(* IEC 61131-3 sources: volt/packages/volt-lsp-iec/test-corpus/bakon-nano/Device/Plc Logic/Application/POUs/RecipeManagement, 4 files *)

(* ---- L_RecipeManager.pou ---- *)
FUNCTION_BLOCK L_RecipeManager
VAR_INPUT
	xEnable					: BOOL;				//Enable functions
	sDatabaseName			: STRING;			//Database of recipe manager (name)
	sRecipeName				: STRING;			//Selected recipe (name)
END_VAR
VAR_IN_OUT
	xRecipe_Delete			: BOOL;				//Delete definition (DeleteRecipeFile)
	xRecipe_Load			: BOOL;				//Load recipe (LoadAndWriteRecipe)
	xRecipe_Save			: BOOL;				//Save recipe (ReadAndSaveRecipe)
	xRecipe_SaveAs			: BOOL;				//Save recipe (ReadAndSaveRecipe)
	sActiveRecipe			: STRING;			//Active machine recipe
END_VAR
VAR_OUTPUT
	xEnabled				: BOOL;				//Function enabled
	iNumberOfRecipes		: INT;				//Counted recipes in database
	sRecipeNames			: STRING(gc_iSizeRecipesNames);	//Combined recipe names
	dwReturnValue			: DWORD;			//Return value of recipe manager
END_VAR

VAR
	RecipeHandler			: RecipeManCommands;//Function to access PLC recipes
	sRecipeLocal			: STRING;			//Used to concat
	psNames					: POINTER TO STRING(gc_iSizeRecipesNames);
	psLocal					: POINTER TO STRING;
	iLoopNames				: INT;				//Loop recipe names
	strSearchChar			: STRING;
	iResult					: INT;
END_VAR
VAR CONSTANT
	gc_iSizeRecipesNames 	: INT := 5000;
	//gc_iMaxResultsFinder	: INT := 10;
END_VAR
%LANGUAGE ST
IF xEnable THEN
	xEnabled := xEnable;
	//************************************************************************Refresh data
	//Get data addresses
	psNames := ADR(sRecipeNames);
	psLocal := ADR(sRecipeLocal);
	//Refresh file buffer
	RecipeHandler.ReloadRecipes(sDatabaseName);
	//Get recipe count
	iNumberOfRecipes := RecipeHandler.GetRecipeCount(sDatabaseName);
	//Get saved recipe informations
	sRecipeNames:='';
	FOR iLoopNames:=0 TO iNumberOfRecipes-1 BY 1 DO
		//Get recipe name
		sRecipeLocal := '';
		RecipeHandler.GetRecipeNames(sDatabaseName, ADR(sRecipeLocal) , 1, iLoopNames);

		//Add recipe name to end of string
		StrConcatA(pstFrom:= psLocal, pstTo:= psNames, iBufferSize:= gc_iSizeRecipesNames);

		//Add seperator to end
		sRecipeLocal := ';';
		StrConcatA(pstFrom:= psLocal, pstTo:= psNames, iBufferSize:= gc_iSizeRecipesNames);
	END_FOR

	//************************************************************************Load recipe to HMI
	IF xRecipe_Load THEN
		dwReturnValue:=RecipeHandler.LoadAndWriteRecipe(sDatabaseName, sRecipeName);//Load to handler recipe
		IF dwReturnValue = 0 THEN
			sActiveRecipe := sRecipeName;
		END_IF
		xRecipe_Load:=FALSE;
	END_IF
	//************************************************************************Save recipe to database
	IF xRecipe_Save THEN
		dwReturnValue:=RecipeHandler.ReadAndSaveRecipe(sDatabaseName, sActiveRecipe);		//Save to file
		xRecipe_Save := FALSE;
	END_IF
	//************************************************************************Delete recipe
	//More than 0 recipes left
	IF xRecipe_Delete THEN
		dwReturnValue:=RecipeHandler.DeleteRecipe(sDatabaseName, sRecipeName);	//Remove database link
		IF sActiveRecipe = sRecipeName THEN
			sActiveRecipe:='';
		END_IF
		xRecipe_Delete := FALSE;
	END_IF
	//************************************************************************Save recipe as
	IF xRecipe_SaveAs THEN
		strSearchChar:='.';
		iResult:=StrFindA(pst1:=ADR(sRecipeName) , pst2:= ADR(strSearchChar), uiSearchStart:= 0);
		IF iResult <> 0 THEN
			dwReturnValue:=16#7000;
			RETURN;
		END_IF

		dwReturnValue:=RecipeHandler.CreateRecipe(sDatabaseName, sRecipeName);		//Create new file and save

		//New recipe OR when recipe already existed
		IF dwReturnValue = 16#4005 OR dwReturnValue = 0 THEN
			dwReturnValue:=RecipeHandler.ReadAndSaveRecipe(sDatabaseName, sRecipeName);	//Create new file and save
		END_IF
		IF dwReturnValue = 0 THEN
			dwReturnValue:=RecipeHandler.LoadAndWriteRecipe(sDatabaseName, sRecipeName);//Load to handler recipe
			dwReturnValue:=SEL(dwReturnValue <> 0, 0, 16#7001);
		END_IF
		IF dwReturnValue = 0 THEN
			sActiveRecipe := sRecipeName;
		END_IF
		xRecipe_SaveAs := FALSE;
	END_IF

ELSE
	sActiveRecipe := '';
	dwReturnValue:=0;
END_IF

END_FUNCTION_BLOCK

(* ---- L_RecipeManager_Rcp.pou ---- *)
FUNCTION_BLOCK L_RecipeManager_Rcp
VAR_INPUT
	xEnable						: BOOL;				//Enable functions
	sDatabaseName				: STRING;			//Database of recipe manager (name)
END_VAR
VAR_IN_OUT
	sSelectedRecipeName			: STRING;
	xRecipe_Load				: BOOL;
	xRecipe_New					: BOOL;
	xRecipe_Edit				: BOOL;
	xRecipe_Save				: BOOL;
	xRecipe_Copy				: BOOL;
	xRecipe_Delete				: BOOL;
	xRecipe_Update				: BOOL;
	scRecipeVisu				: sMACH_RCP_Parameters;
	scRecipePLC					: sMACH_RCP_Parameters;
END_VAR
VAR_OUTPUT
	xEnabled					: BOOL;				//Function enabled
	iNumberOfRecipes			: INT;				//Counted recipes in database
	sRecipeNames				: STRING(gc_iSizeRecipesNames);	//Combined recipe names
	dwReturnValue				: DWORD;			//Return value of recipe manager
END_VAR
VAR
	RecipeHandler				: RecipeManCommands;//Function to access PLC recipes
	sRecipeLocal				: STRING;			//Used to concat
	psNames						: POINTER TO STRING(gc_iSizeRecipesNames);
	psLocal						: POINTER TO STRING;
	iLoopNames					: INT;				//Loop recipe names
	strSearchChar				: STRING;
	iResult						: INT;
	sRecipNameTemp: STRING;
END_VAR
VAR CONSTANT
	gc_iSizeRecipesNames 		: INT := 16384;
END_VAR
%LANGUAGE ST
IF xEnable THEN
	xEnabled := xEnable;
	//************************************************************************Refresh data
	//Get data addresses
	psNames := ADR(sRecipeNames);
	psLocal := ADR(sRecipeLocal);
	//Refresh file buffer
	RecipeHandler.ReloadRecipes(sDatabaseName);
	//Get recipe count
	iNumberOfRecipes := RecipeHandler.GetRecipeCount(sDatabaseName);
	//Get saved recipe informations
	sRecipeNames:='';
	FOR iLoopNames:=0 TO iNumberOfRecipes-1 BY 1 DO
		//Get recipe name
		sRecipeLocal := '';
		RecipeHandler.GetRecipeNames(sDatabaseName, ADR(sRecipeLocal) , 1, iLoopNames);

		//Add recipe name to end of string
		StrConcatA(pstFrom:= psLocal, pstTo:= psNames, iBufferSize:= gc_iSizeRecipesNames);

		//Add seperator to end
		sRecipeLocal := ';';
		StrConcatA(pstFrom:= psLocal, pstTo:= psNames, iBufferSize:= gc_iSizeRecipesNames);
	END_FOR
	IF xRecipe_Load THEN
		dwReturnValue:=RecipeHandler.LoadAndWriteRecipe(sDatabaseName, sSelectedRecipeName);//Load to handler recipe
		IF dwReturnValue = 0 THEN
			scRecipePLC:=scRecipeVisu;
		END_IF
		xRecipe_Load:=FALSE;
	END_IF
	IF xRecipe_New THEN
		strSearchChar:='.';
		dwReturnValue:=INT_TO_DWORD(StrFindA(pst1:=ADR(scRecipeVisu.sRecipeName) , pst2:= ADR(strSearchChar), uiSearchStart:= 0));
		IF dwReturnValue = 0 THEN
			dwReturnValue:=RecipeHandler.CreateRecipe(sDatabaseName, scRecipeVisu.sRecipeName);
		ELSE
			dwReturnValue:=16#7000;
		END_IF
		xRecipe_New := FALSE;
	END_IF
	IF xRecipe_Edit THEN
		dwReturnValue:=RecipeHandler.LoadAndWriteRecipe(sDatabaseName, sSelectedRecipeName);//Load to handler recipe
		xRecipe_Edit:=FALSE;
	END_IF
	IF xRecipe_Save THEN
		dwReturnValue:=RecipeHandler.ReadAndSaveRecipe(sDatabaseName, scRecipeVisu.sRecipeName);	//Create new file and save
		xRecipe_Save := FALSE;
	END_IF
	IF xRecipe_Copy THEN
		sRecipNameTemp:=scRecipeVisu.sRecipeName;
		dwReturnValue:=RecipeHandler.LoadAndWriteRecipe(sDatabaseName, sSelectedRecipeName);
		scRecipeVisu.sRecipeName:=sRecipNameTemp;
		strSearchChar:='.';
		dwReturnValue:=INT_TO_DWORD(StrFindA(pst1:=ADR(scRecipeVisu.sRecipeName) , pst2:= ADR(strSearchChar), uiSearchStart:= 0));
		IF dwReturnValue = 0 THEN
			dwReturnValue:=RecipeHandler.CreateRecipe(sDatabaseName, scRecipeVisu.sRecipeName);
		ELSE
			dwReturnValue:=16#7000;
		END_IF
		xRecipe_Copy := FALSE;
	END_IF
	IF xRecipe_Delete THEN
		dwReturnValue:=RecipeHandler.DeleteRecipe(sDatabaseName, sSelectedRecipeName);	//Remove database link
		xRecipe_Delete := FALSE;
	END_IF
	IF xRecipe_Update THEN
		scRecipeVisu:=scRecipePLC;
		dwReturnValue:=RecipeHandler.ReadAndSaveRecipe(sDatabaseName, scRecipeVisu.sRecipeName);	//Create new file and save
		xRecipe_Update := FALSE;
	END_IF
ELSE
	dwReturnValue:=0;
END_IF

END_FUNCTION_BLOCK

(* ---- RCP_RecipeHandler.pou ---- *)
PROGRAM RCP_RecipeHandler
VAR
	{warning 'Disabled for compatibility SVE'}
	//DiffLogger								: DifferenceLogger;
	bOldRect : BOOL;
	bOldEight : BOOL;
END_VAR
%LANGUAGE ST
(*Reset recipe*)
IF		g_HMI_MachCommand.CMD.bResetRecipe
THEN

		g_HMI_RCP_Parameters.nProductType				:= Prod_Tray_Rectangle_1x1;
		g_HMI_RCP_Parameters.rStartHeightKnife			:= 60;		(* Starthoogte, gemeten vanaf onderzijde mes tot aan de tafel *)
		g_HMI_RCP_Parameters.rStopHeightKnife			:= 0;		(* Stophoogte, gemeten vanaf onderzijde mes tot aan de tafel *)
		g_HMI_RCP_Parameters.nPartsRound				:= 12;			(*aantal stukken ronde taart *)
		g_HMI_RCP_Parameters.nPartsX					:= 5;			(*aantal stukken in X richting*)
		g_HMI_RCP_Parameters.nPartsY					:= 5;			(*aantal stukken in Y richting*)
		g_HMI_RCP_Parameters.rAngleInDegrees			:= 55;		(* Angle in degrees when producttype is diagonal *)
		g_HMI_RCP_Parameters.rProdLength_InX			:= 500;		(* Size of slab in line with the belt*)
		g_HMI_RCP_Parameters.rProdLength_InY			:= 300;		(* Size of slab perpendicular to the belt*)
		g_HMI_RCP_Parameters.rUSHeightStart			:= 60;		(* Start height ultrasonic generator (position Z-axis) *)
		g_HMI_RCP_Parameters.rUSHeightStop			:= 60;		(* Stop height ultrasonic generator (position Z-axis) *)
		g_HMI_RCP_Parameters.dwUltrasonicPower1		:= 50;
		g_HMI_RCP_Parameters.rCutSpeedZ_Down1		:= 50;			(* neergaande snelheid boven product in %*)
		g_HMI_RCP_Parameters.rCutSpeedZ_Down2		:= 50;			(* neergaande snelheid in het product in %*)
		g_HMI_RCP_Parameters.rCutSpeedZ_Up1			:= 50;			(* opgaande snelheid in het product in %*)
		g_HMI_RCP_Parameters.rSizeTrimRight			:= 8;		(*grootte van de afvalrand in de X richting aan de rechterzijde*)
		g_HMI_RCP_Parameters.rSizeTrimLeft			:= 8;		(*grootte van de afvalrand in de X richting aan de linkerzijde*)
		g_HMI_RCP_Parameters.rSizeTrimRear				:= 8;		(*grootte van de afvalrand in de Y richting aan de achterzijde*)
		g_HMI_RCP_Parameters.rSizeTrimFront			:= 8;		(*grootte van de afvalrand in de Y richting aan de voorzijde*)
		g_HMI_RCP_Parameters.rMidPosOffsetRound1X	:= 0;		(* For round products *)
		g_HMI_RCP_Parameters.rMidPosOffsetRound1Y	:= 0;		(* For round products *)
		g_HMI_RCP_Parameters.rMidPosOffsetRound2X	:= 0;		(* For round products *)
		g_HMI_RCP_Parameters.rMidPosOffsetRound2Y	:= 0;		(* For round products *)
		g_HMI_RCP_Parameters.bUseRectanglesForTriangles	:= FALSE;	(* For triangles only *)
		g_HMI_RCP_Parameters.rPartSizeX					:= 50;		(* For triangles only *)
		g_HMI_RCP_Parameters.rPartSizeY					:= 50;		(* For triangles only *)
		g_HMI_RCP_Parameters.rShiftCompensation		:= 0;

		g_HMI_MachCommand.CMD.bResetRecipe		:= FALSE;
		g_HMI_bRecipeIsReset								:= TRUE;

END_IF

(* Recept variabele driehoek in tray resetten indien deze keuze niet gemaakt is in de product optie pagina *)
IF NOT g_HMI_dwProductOptions.15 THEN
	g_HMI_RCP_Parameters.bTrianglesInTray := FALSE;
END_IF

(*Afvalrand limieten bepalen*) (*Minimaal een stuk van 10mm overhouden, maximale afvalrand van 500*)
CASE G_HMI_RCP_Parameters.nProductType OF
	Prod_Slab_Rectangle_1x1, Prod_Slab_Triangle_1x1, Prod_Slab_Diagonal_1x1, Prod_Slab_Rectangle_1x1_Clamp:	(*Slab products*)
	g_sHMI_Mach_UnitStatus.rWasteFrontMax 	:= MIN(500,(g_HMI_RCP_Parameters.rProdLength_InY - 10 - g_HMI_RCP_Parameters.rSizeTrimRear));
	g_sHMI_Mach_UnitStatus.rWasteRearMax 	:= MIN(500,(g_HMI_RCP_Parameters.rProdLength_InY - 10 - g_HMI_RCP_Parameters.rSizeTrimFront));
	g_sHMI_Mach_UnitStatus.rWasteRightMax 	:= MIN(500,(g_HMI_RCP_Parameters.rProdLength_InX - 10 - g_HMI_RCP_Parameters.rSizeTrimLeft));
	g_sHMI_Mach_UnitStatus.rWasteLeftMax 	:= MIN(500,(g_HMI_RCP_Parameters.rProdLength_InX - 10 - g_HMI_RCP_Parameters.rSizeTrimRight));

	Prod_Tray_Rectangle_1x2		:		(* ProductType = 4 = Tray Square Small *)
	g_sHMI_Mach_UnitStatus.rWasteFrontMax 	:= MIN(500,(g_HMI_MCH_Parameters.rProdLengthTraySmall_InY - 10 - g_HMI_RCP_Parameters.rSizeTrimRear));
	g_sHMI_Mach_UnitStatus.rWasteRearMax 	:= MIN(500,(g_HMI_MCH_Parameters.rProdLengthTraySmall_InY - 10 - g_HMI_RCP_Parameters.rSizeTrimFront));
	g_sHMI_Mach_UnitStatus.rWasteRightMax 	:= MIN(500,(g_HMI_MCH_Parameters.rProdLengthTraySmall_InX - 10 - g_HMI_RCP_Parameters.rSizeTrimLeft));
	g_sHMI_Mach_UnitStatus.rWasteLeftMax 	:= MIN(500,(g_HMI_MCH_Parameters.rProdLengthTraySmall_InX - 10 - g_HMI_RCP_Parameters.rSizeTrimRight));

	Prod_Tray_Rectangle_1x1		:		(* ProductType = 5 = Tray Square Large *)
	g_sHMI_Mach_UnitStatus.rWasteFrontMax 	:= MIN(500,(g_HMI_MCH_Parameters.rProdLengthTrayLarge_InY - 10 - g_HMI_RCP_Parameters.rSizeTrimRear));
	g_sHMI_Mach_UnitStatus.rWasteRearMax 	:= MIN(500,(g_HMI_MCH_Parameters.rProdLengthTrayLarge_InY - 10 - g_HMI_RCP_Parameters.rSizeTrimFront));
	g_sHMI_Mach_UnitStatus.rWasteRightMax 	:= MIN(500,(g_HMI_MCH_Parameters.rProdLengthTrayLarge_InX - 10 - g_HMI_RCP_Parameters.rSizeTrimLeft));
	g_sHMI_Mach_UnitStatus.rWasteLeftMax 	:= MIN(500,(g_HMI_MCH_Parameters.rProdLengthTrayLarge_InX - 10 - g_HMI_RCP_Parameters.rSizeTrimRight));

	Prod_Tray_Rectangle_1x4		:		(* ProductType = 6 = Tray Square 4 on a table *)
	g_sHMI_Mach_UnitStatus.rWasteFrontMax 	:= MIN(500,(g_HMI_MCH_Parameters.rProdLengthTrayTriple_InY - 10 - g_HMI_RCP_Parameters.rSizeTrimRear));
	g_sHMI_Mach_UnitStatus.rWasteRearMax 	:= MIN(500,(g_HMI_MCH_Parameters.rProdLengthTrayTriple_InY - 10 - g_HMI_RCP_Parameters.rSizeTrimFront));
	g_sHMI_Mach_UnitStatus.rWasteRightMax 	:= MIN(500,(g_HMI_MCH_Parameters.rProdLengthTrayTriple_InX - 10 - g_HMI_RCP_Parameters.rSizeTrimLeft));
	g_sHMI_Mach_UnitStatus.rWasteLeftMax 	:= MIN(500,(g_HMI_MCH_Parameters.rProdLengthTrayTriple_InX - 10 - g_HMI_RCP_Parameters.rSizeTrimRight));

	Prod_Tray_Rectangle_2x1		:		(* ProductType = 8 = Tray square 2 side by side*)
	g_sHMI_Mach_UnitStatus.rWasteFrontMax 	:= MIN(500,(g_HMI_MCH_Parameters.rProdLengthTrayDouble_InY - 10 - g_HMI_RCP_Parameters.rSizeTrimRear));
	g_sHMI_Mach_UnitStatus.rWasteRearMax 	:= MIN(500,(g_HMI_MCH_Parameters.rProdLengthTrayDouble_InY - 10 - g_HMI_RCP_Parameters.rSizeTrimFront));
	g_sHMI_Mach_UnitStatus.rWasteRightMax 	:= MIN(500,(g_HMI_MCH_Parameters.rProdLengthTrayDouble_InX - 10 - g_HMI_RCP_Parameters.rSizeTrimLeft));
	g_sHMI_Mach_UnitStatus.rWasteLeftMax 	:= MIN(500,(g_HMI_MCH_Parameters.rProdLengthTrayDouble_InX - 10 - g_HMI_RCP_Parameters.rSizeTrimRight));

END_CASE

(*Minimale Afvalrand limieten bepalen*)
CASE G_HMI_RCP_Parameters.nProductType OF
	Prod_Slab_Rectangle_1x1, Prod_Slab_Triangle_1x1, Prod_Slab_Diagonal_1x1, Prod_Slab_Rectangle_1x1_Clamp:	(*Slab products*)
	g_sHMI_Mach_UnitStatus.rWasteFrontMin 	:= 0; // was -50;
	g_sHMI_Mach_UnitStatus.rWasteRearMin 	:= 0; // was -50;
	g_sHMI_Mach_UnitStatus.rWasteRightMin 	:= 0; // was -50;
	g_sHMI_Mach_UnitStatus.rWasteLeftMin 	:= 0; // was -50;

	Prod_Tray_Rectangle_1x2, Prod_Tray_Rectangle_1x1, Prod_Tray_Rectangle_1x4, Prod_Tray_Rectangle_2x1 :	(* Tray products *)
	g_sHMI_Mach_UnitStatus.rWasteFrontMin 	:= 0;
	g_sHMI_Mach_UnitStatus.rWasteRearMin 	:= 0;
	g_sHMI_Mach_UnitStatus.rWasteRightMin 	:= 0;
	g_sHMI_Mach_UnitStatus.rWasteLeftMin 	:= 0;
END_CASE

(* Recept variabele driehoek in tray resetten indien deze keuze niet gemaakt is in de product optie pagina *)
IF NOT g_HMI_dwProductOptions.15 THEN
	g_HMI_RCP_Parameters.bTrianglesInTray := FALSE;
END_IF

(*Functioneren van checkboxes als radioboxes*)
IF g_HMI_RCP_Parameters.bUseRectanglesForTriangles AND bOldEight THEN
	g_HMI_RCP_Parameters.bUseRectanglesInEight := FALSE;
END_IF

IF g_HMI_RCP_Parameters.bUseRectanglesInEight AND bOldRect THEN
	g_HMI_RCP_Parameters.bUseRectanglesForTriangles := FALSE;
END_IF

bOldEight := g_HMI_RCP_Parameters.bUseRectanglesInEight;
bOldRect := g_HMI_RCP_Parameters.bUseRectanglesForTriangles;

IF NOT g_sRCPCopyMade THEN
	g_sRCPParCopy := g_HMI_RCP_Parameters;
	g_sRCPCopyMade	:= TRUE;
END_IF

(*DiffLogger.orig := __VARINFO(g_HMI_RCP_Parameters.nProductType); DiffLogger.copy := __VARINFO(               g_sRCPParCopy.nProductType); DiffLogger(	Logger := ADR(g_Logger), copyStr := TO_STRING(               g_sRCPParCopy.nProductType), origStr := TO_STRING(g_HMI_RCP_Parameters.nProductType));
DiffLogger.orig := __VARINFO(g_HMI_RCP_Parameters.rStartHeightKnife); DiffLogger.copy := __VARINFO(          g_sRCPParCopy.rStartHeightKnife); DiffLogger(	Logger := ADR(g_Logger), copyStr := TO_STRING(          g_sRCPParCopy.rStartHeightKnife), origStr := TO_STRING(g_HMI_RCP_Parameters.rStartHeightKnife));
DiffLogger.orig := __VARINFO(g_HMI_RCP_Parameters.rStopHeightKnife); DiffLogger.copy := __VARINFO(           g_sRCPParCopy.rStopHeightKnife); DiffLogger(	Logger := ADR(g_Logger), copyStr := TO_STRING(           g_sRCPParCopy.rStopHeightKnife), origStr := TO_STRING(g_HMI_RCP_Parameters.rStopHeightKnife));
DiffLogger.orig := __VARINFO(g_HMI_RCP_Parameters.nPartsRound); DiffLogger.copy := __VARINFO(                g_sRCPParCopy.nPartsRound); DiffLogger(	Logger := ADR(g_Logger), copyStr := TO_STRING(                g_sRCPParCopy.nPartsRound), origStr := TO_STRING(g_HMI_RCP_Parameters.nPartsRound));
DiffLogger.orig := __VARINFO(g_HMI_RCP_Parameters.nPartsRoundRight); DiffLogger.copy := __VARINFO(           g_sRCPParCopy.nPartsRoundRight); DiffLogger(	Logger := ADR(g_Logger), copyStr := TO_STRING(           g_sRCPParCopy.nPartsRoundRight), origStr := TO_STRING(g_HMI_RCP_Parameters.nPartsRoundRight));
DiffLogger.orig := __VARINFO(g_HMI_RCP_Parameters.nPartsX); DiffLogger.copy := __VARINFO(                    g_sRCPParCopy.nPartsX); DiffLogger(	Logger := ADR(g_Logger), copyStr := TO_STRING(                    g_sRCPParCopy.nPartsX), origStr := TO_STRING(g_HMI_RCP_Parameters.nPartsX));
DiffLogger.orig := __VARINFO(g_HMI_RCP_Parameters.nPartsY); DiffLogger.copy := __VARINFO(                    g_sRCPParCopy.nPartsY); DiffLogger(	Logger := ADR(g_Logger), copyStr := TO_STRING(                    g_sRCPParCopy.nPartsY), origStr := TO_STRING(g_HMI_RCP_Parameters.nPartsY));
DiffLogger.orig := __VARINFO(g_HMI_RCP_Parameters.rAngleInDegrees); DiffLogger.copy := __VARINFO(            g_sRCPParCopy.rAngleInDegrees); DiffLogger(	Logger := ADR(g_Logger), copyStr := TO_STRING(            g_sRCPParCopy.rAngleInDegrees), origStr := TO_STRING(g_HMI_RCP_Parameters.rAngleInDegrees));
DiffLogger.orig := __VARINFO(g_HMI_RCP_Parameters.rProdLength_InX); DiffLogger.copy := __VARINFO(            g_sRCPParCopy.rProdLength_InX); DiffLogger(	Logger := ADR(g_Logger), copyStr := TO_STRING(            g_sRCPParCopy.rProdLength_InX), origStr := TO_STRING(g_HMI_RCP_Parameters.rProdLength_InX));
DiffLogger.orig := __VARINFO(g_HMI_RCP_Parameters.rProdLength_InY); DiffLogger.copy := __VARINFO(            g_sRCPParCopy.rProdLength_InY); DiffLogger(	Logger := ADR(g_Logger), copyStr := TO_STRING(            g_sRCPParCopy.rProdLength_InY), origStr := TO_STRING(g_HMI_RCP_Parameters.rProdLength_InY));
DiffLogger.orig := __VARINFO(g_HMI_RCP_Parameters.rUSHeightStart); DiffLogger.copy := __VARINFO(             g_sRCPParCopy.rUSHeightStart); DiffLogger(	Logger := ADR(g_Logger), copyStr := TO_STRING(             g_sRCPParCopy.rUSHeightStart), origStr := TO_STRING(g_HMI_RCP_Parameters.rUSHeightStart));
DiffLogger.orig := __VARINFO(g_HMI_RCP_Parameters.rUSHeightStop); DiffLogger.copy := __VARINFO(              g_sRCPParCopy.rUSHeightStop); DiffLogger(	Logger := ADR(g_Logger), copyStr := TO_STRING(              g_sRCPParCopy.rUSHeightStop), origStr := TO_STRING(g_HMI_RCP_Parameters.rUSHeightStop));
DiffLogger.orig := __VARINFO(g_HMI_RCP_Parameters.dwUltrasonicPower1); DiffLogger.copy := __VARINFO(         g_sRCPParCopy.dwUltrasonicPower1); DiffLogger(	Logger := ADR(g_Logger), copyStr := TO_STRING(         g_sRCPParCopy.dwUltrasonicPower1), origStr := TO_STRING(g_HMI_RCP_Parameters.dwUltrasonicPower1));
DiffLogger.orig := __VARINFO(g_HMI_RCP_Parameters.rCutSpeedZ_Down1); DiffLogger.copy := __VARINFO(           g_sRCPParCopy.rCutSpeedZ_Down1); DiffLogger(	Logger := ADR(g_Logger), copyStr := TO_STRING(           g_sRCPParCopy.rCutSpeedZ_Down1), origStr := TO_STRING(g_HMI_RCP_Parameters.rCutSpeedZ_Down1));
DiffLogger.orig := __VARINFO(g_HMI_RCP_Parameters.rCutSpeedZ_Down2); DiffLogger.copy := __VARINFO(           g_sRCPParCopy.rCutSpeedZ_Down2); DiffLogger(	Logger := ADR(g_Logger), copyStr := TO_STRING(           g_sRCPParCopy.rCutSpeedZ_Down2), origStr := TO_STRING(g_HMI_RCP_Parameters.rCutSpeedZ_Down2));
DiffLogger.orig := __VARINFO(g_HMI_RCP_Parameters.rCutSpeedZ_Up1); DiffLogger.copy := __VARINFO(             g_sRCPParCopy.rCutSpeedZ_Up1); DiffLogger(	Logger := ADR(g_Logger), copyStr := TO_STRING(             g_sRCPParCopy.rCutSpeedZ_Up1), origStr := TO_STRING(g_HMI_RCP_Parameters.rCutSpeedZ_Up1));
DiffLogger.orig := __VARINFO(g_HMI_RCP_Parameters.rSizeTrimRight); DiffLogger.copy := __VARINFO(             g_sRCPParCopy.rSizeTrimRight); DiffLogger(	Logger := ADR(g_Logger), copyStr := TO_STRING(             g_sRCPParCopy.rSizeTrimRight), origStr := TO_STRING(g_HMI_RCP_Parameters.rSizeTrimRight));
DiffLogger.orig := __VARINFO(g_HMI_RCP_Parameters.rSizeTrimLeft); DiffLogger.copy := __VARINFO(              g_sRCPParCopy.rSizeTrimLeft); DiffLogger(	Logger := ADR(g_Logger), copyStr := TO_STRING(              g_sRCPParCopy.rSizeTrimLeft), origStr := TO_STRING(g_HMI_RCP_Parameters.rSizeTrimLeft));
DiffLogger.orig := __VARINFO(g_HMI_RCP_Parameters.rSizeTrimRear); DiffLogger.copy := __VARINFO(              g_sRCPParCopy.rSizeTrimRear); DiffLogger(	Logger := ADR(g_Logger), copyStr := TO_STRING(              g_sRCPParCopy.rSizeTrimRear), origStr := TO_STRING(g_HMI_RCP_Parameters.rSizeTrimRear));
DiffLogger.orig := __VARINFO(g_HMI_RCP_Parameters.rSizeTrimFront); DiffLogger.copy := __VARINFO(             g_sRCPParCopy.rSizeTrimFront); DiffLogger(	Logger := ADR(g_Logger), copyStr := TO_STRING(             g_sRCPParCopy.rSizeTrimFront), origStr := TO_STRING(g_HMI_RCP_Parameters.rSizeTrimFront));
DiffLogger.orig := __VARINFO(g_HMI_RCP_Parameters.rDiameterRound); DiffLogger.copy := __VARINFO(             g_sRCPParCopy.rDiameterRound); DiffLogger(	Logger := ADR(g_Logger), copyStr := TO_STRING(             g_sRCPParCopy.rDiameterRound), origStr := TO_STRING(g_HMI_RCP_Parameters.rDiameterRound));
DiffLogger.orig := __VARINFO(g_HMI_RCP_Parameters.rMidPosOffsetRound1X); DiffLogger.copy := __VARINFO(       g_sRCPParCopy.rMidPosOffsetRound1X); DiffLogger(	Logger := ADR(g_Logger), copyStr := TO_STRING(       g_sRCPParCopy.rMidPosOffsetRound1X), origStr := TO_STRING(g_HMI_RCP_Parameters.rMidPosOffsetRound1X));
DiffLogger.orig := __VARINFO(g_HMI_RCP_Parameters.rMidPosOffsetRound1Y); DiffLogger.copy := __VARINFO(       g_sRCPParCopy.rMidPosOffsetRound1Y); DiffLogger(	Logger := ADR(g_Logger), copyStr := TO_STRING(       g_sRCPParCopy.rMidPosOffsetRound1Y), origStr := TO_STRING(g_HMI_RCP_Parameters.rMidPosOffsetRound1Y));
DiffLogger.orig := __VARINFO(g_HMI_RCP_Parameters.rMidPosOffsetRound2X); DiffLogger.copy := __VARINFO(       g_sRCPParCopy.rMidPosOffsetRound2X); DiffLogger(	Logger := ADR(g_Logger), copyStr := TO_STRING(       g_sRCPParCopy.rMidPosOffsetRound2X), origStr := TO_STRING(g_HMI_RCP_Parameters.rMidPosOffsetRound2X));
DiffLogger.orig := __VARINFO(g_HMI_RCP_Parameters.rMidPosOffsetRound2Y); DiffLogger.copy := __VARINFO(       g_sRCPParCopy.rMidPosOffsetRound2Y); DiffLogger(	Logger := ADR(g_Logger), copyStr := TO_STRING(       g_sRCPParCopy.rMidPosOffsetRound2Y), origStr := TO_STRING(g_HMI_RCP_Parameters.rMidPosOffsetRound2Y));
DiffLogger.orig := __VARINFO(g_HMI_RCP_Parameters.bTrianglesInTray); DiffLogger.copy := __VARINFO(           g_sRCPParCopy.bTrianglesInTray); DiffLogger(	Logger := ADR(g_Logger), copyStr := TO_STRING(           g_sRCPParCopy.bTrianglesInTray), origStr := TO_STRING(g_HMI_RCP_Parameters.bTrianglesInTray));
DiffLogger.orig := __VARINFO(g_HMI_RCP_Parameters.bUseRectanglesForTriangles); DiffLogger.copy := __VARINFO( g_sRCPParCopy.bUseRectanglesForTriangles); DiffLogger(	Logger := ADR(g_Logger), copyStr := TO_STRING( g_sRCPParCopy.bUseRectanglesForTriangles), origStr := TO_STRING(g_HMI_RCP_Parameters.bUseRectanglesForTriangles));
DiffLogger.orig := __VARINFO(g_HMI_RCP_Parameters.bUseRectanglesInEight); DiffLogger.copy := __VARINFO(      g_sRCPParCopy.bUseRectanglesInEight); DiffLogger(	Logger := ADR(g_Logger), copyStr := TO_STRING(      g_sRCPParCopy.bUseRectanglesInEight), origStr := TO_STRING(g_HMI_RCP_Parameters.bUseRectanglesInEight));
DiffLogger.orig := __VARINFO(g_HMI_RCP_Parameters.bCutRoundInSequence); DiffLogger.copy := __VARINFO(        g_sRCPParCopy.bCutRoundInSequence); DiffLogger(	Logger := ADR(g_Logger), copyStr := TO_STRING(        g_sRCPParCopy.bCutRoundInSequence), origStr := TO_STRING(g_HMI_RCP_Parameters.bCutRoundInSequence));
DiffLogger.orig := __VARINFO(g_HMI_RCP_Parameters.bCutWasteFirst); DiffLogger.copy := __VARINFO(             g_sRCPParCopy.bCutWasteFirst); DiffLogger(	Logger := ADR(g_Logger), copyStr := TO_STRING(             g_sRCPParCopy.bCutWasteFirst), origStr := TO_STRING(g_HMI_RCP_Parameters.bCutWasteFirst));
DiffLogger.orig := __VARINFO(g_HMI_RCP_Parameters.rPartSizeX); DiffLogger.copy := __VARINFO(                 g_sRCPParCopy.rPartSizeX); DiffLogger(	Logger := ADR(g_Logger), copyStr := TO_STRING(                 g_sRCPParCopy.rPartSizeX), origStr := TO_STRING(g_HMI_RCP_Parameters.rPartSizeX));
DiffLogger.orig := __VARINFO(g_HMI_RCP_Parameters.rPartSizeY); DiffLogger.copy := __VARINFO(                 g_sRCPParCopy.rPartSizeY); DiffLogger(	Logger := ADR(g_Logger), copyStr := TO_STRING(                 g_sRCPParCopy.rPartSizeY), origStr := TO_STRING(g_HMI_RCP_Parameters.rPartSizeY));
DiffLogger.orig := __VARINFO(g_HMI_RCP_Parameters.rShiftCompensation); DiffLogger.copy := __VARINFO(         g_sRCPParCopy.rShiftCompensation); DiffLogger(	Logger := ADR(g_Logger), copyStr := TO_STRING(         g_sRCPParCopy.rShiftCompensation), origStr := TO_STRING(g_HMI_RCP_Parameters.rShiftCompensation));
DiffLogger.orig := __VARINFO(g_HMI_RCP_Parameters.rSpeedTableXY); DiffLogger.copy := __VARINFO(              g_sRCPParCopy.rSpeedTableXY); DiffLogger(	Logger := ADR(g_Logger), copyStr := TO_STRING(              g_sRCPParCopy.rSpeedTableXY), origStr := TO_STRING(g_HMI_RCP_Parameters.rSpeedTableXY));
DiffLogger.orig := __VARINFO(g_HMI_RCP_Parameters.rCleaningTimeUltrasonic); DiffLogger.copy := __VARINFO(    g_sRCPParCopy.rCleaningTimeUltrasonic); DiffLogger(	Logger := ADR(g_Logger), copyStr := TO_STRING(    g_sRCPParCopy.rCleaningTimeUltrasonic), origStr := TO_STRING(g_HMI_RCP_Parameters.rCleaningTimeUltrasonic));
DiffLogger.orig := __VARINFO(g_HMI_RCP_Parameters.rCleaningTimeWater); DiffLogger.copy := __VARINFO(         g_sRCPParCopy.rCleaningTimeWater); DiffLogger(	Logger := ADR(g_Logger), copyStr := TO_STRING(         g_sRCPParCopy.rCleaningTimeWater), origStr := TO_STRING(g_HMI_RCP_Parameters.rCleaningTimeWater));
DiffLogger.orig := __VARINFO(g_HMI_RCP_Parameters.rCleaningTimeAir); DiffLogger.copy := __VARINFO(           g_sRCPParCopy.rCleaningTimeAir); DiffLogger(	Logger := ADR(g_Logger), copyStr := TO_STRING(           g_sRCPParCopy.rCleaningTimeAir), origStr := TO_STRING(g_HMI_RCP_Parameters.rCleaningTimeAir));
DiffLogger.orig := __VARINFO(g_HMI_RCP_Parameters.nCleanAfterNProd); DiffLogger.copy := __VARINFO(           g_sRCPParCopy.nCleanAfterNProd); DiffLogger(	Logger := ADR(g_Logger), copyStr := TO_STRING(           g_sRCPParCopy.nCleanAfterNProd), origStr := TO_STRING(g_HMI_RCP_Parameters.nCleanAfterNProd));
DiffLogger.orig := __VARINFO(g_HMI_RCP_Parameters.nCleanProdOrCuts); DiffLogger.copy := __VARINFO(           g_sRCPParCopy.nCleanProdOrCuts); DiffLogger(	Logger := ADR(g_Logger), copyStr := TO_STRING(           g_sRCPParCopy.nCleanProdOrCuts), origStr := TO_STRING(g_HMI_RCP_Parameters.nCleanProdOrCuts));
DiffLogger.orig := __VARINFO(g_HMI_RCP_Parameters.nCleanWithScraper); DiffLogger.copy := __VARINFO(          g_sRCPParCopy.nCleanWithScraper); DiffLogger(	Logger := ADR(g_Logger), copyStr := TO_STRING(          g_sRCPParCopy.nCleanWithScraper), origStr := TO_STRING(g_HMI_RCP_Parameters.nCleanWithScraper));
DiffLogger.orig := __VARINFO(g_HMI_RCP_Parameters.bMirrorDiagonals); DiffLogger.copy := __VARINFO(           g_sRCPParCopy.bMirrorDiagonals); DiffLogger(	Logger := ADR(g_Logger), copyStr := TO_STRING(           g_sRCPParCopy.bMirrorDiagonals), origStr := TO_STRING(g_HMI_RCP_Parameters.bMirrorDiagonals));
*)

END_PROGRAM

(* ---- Recipes.pou ---- *)
PROGRAM Recipes
VAR
	bSaveParAs	: BOOL;
	dtDateTime : DT;
	//Recipe Vars
	L_RecipeManager1: L_RecipeManager_Rcp;
	{attribute 'symbol':='readwrite'}
	sSelectedRecipeName: STRING;
	{attribute 'symbol':='readwrite'}
	dwReturnValue: DWORD;
	{attribute 'symbol':='readwrite'}
	sRecipeNames: STRING(5000);
	{attribute 'symbol':='readwrite'}
	sActiveRecipe: STRING;				// Recommended to make Retain
	//
	//MachPar Vars
	L_MachParManager1: L_RecipeManager;
	{attribute 'symbol':='readwrite'}
	sMachParName: STRING;
	{attribute 'symbol':='readwrite'}
	sMachParNames: STRING(5000);
	{attribute 'symbol':='readwrite'}
	sActiveMachPar: STRING;				// Recommended to make Retain
	{attribute 'symbol':='readwrite'}
	dwMachParReturnValue: DWORD;
	bSavePars	: BOOL;
	sParGeneratedName	: STRING;
	GetDateAndTime: rtclk.GetDateAndTime;

	dtDateAndTIme: DATE_AND_TIME;
	sDateAndTIme: STRING;
	sDateAndTIme1: STRING(255);
	sDateAndTIme2: STRING(255);
	sRecipeNamePar: STRING(255);
END_VAR
%LANGUAGE FBD
%NETWORK
EXECUTE(EN := TRUE, 'IF g_HMI_MachCommand.CMD.bNewRecipe THEN
	g_HMI_RCP_Parameters_Visu.nProductType:=0;			(* ProductType = 0 = Slab Square *)
															(* ProductType = 1 = Slab triangle *)
															(* ProductType = 2 = Slab diagonal *)
															(* ProductType = 3 = Round Cake *)
															(* ProductType = 4 = Tray Square Small *)
															(* ProductType = 5 = Tray Square Large *)

	g_HMI_RCP_Parameters_Visu.rStartHeightKnife := 60;		(* Starthoogte, gemeten vanaf onderzijde mes tot aan de tafel *)
	g_HMI_RCP_Parameters_Visu.rStopHeightKnife:= 0;		(* Stophoogte, gemeten vanaf onderzijde mes tot aan de tafel *)
	g_HMI_RCP_Parameters_Visu.nPartsRound	:= 12;			(*aantal stukken ronde taart *)
	g_HMI_RCP_Parameters_Visu.nPartsRoundRight:= 12;			(*aantal stukken ronde taart op rechter positie*)
	g_HMI_RCP_Parameters_Visu.nPartsX	:= 5;			(*aantal stukken in X richting*)
	g_HMI_RCP_Parameters_Visu.nPartsY:= 5;			(*aantal stukken in Y richting*)
	g_HMI_RCP_Parameters_Visu.rAngleInDegrees	 := 40;		(* Angle in degrees when producttype is diagonal *)
	g_HMI_RCP_Parameters_Visu.rProdLength_InX	:=600;
	g_HMI_RCP_Parameters_Visu.rProdLength_InY	:=400;
	g_HMI_RCP_Parameters_Visu.rUSHeightStart:= 60;		(* Start height ultrasonic generator (position Z-axis) *)
	g_HMI_RCP_Parameters_Visu.rUSHeightStop:= 60;		(* Stop height ultrasonic generator (position Z-axis) *)
	g_HMI_RCP_Parameters_Visu.dwUltrasonicPower1:=50;
	g_HMI_RCP_Parameters_Visu.rCutSpeedZ_Down1:=50;			(* neergaande snelheid boven product in %*)
	g_HMI_RCP_Parameters_Visu.rCutSpeedZ_Down2:=50;			(* neergaande snelheid in het product in %*)
	g_HMI_RCP_Parameters_Visu.rCutSpeedZ_Up1:=50;			(* opgaande snelheid in het product in %*)
	g_HMI_RCP_Parameters_Visu.rSizeTrimRight:=60;		(*grootte van de afvalrand in de X richting aan de voorzijde*)
	g_HMI_RCP_Parameters_Visu.rSizeTrimLeft:=60;		(*grootte van de afvalrand in de X richting aan de achterzijde*)
	g_HMI_RCP_Parameters_Visu.rSizeTrimRear:=60;		(*grootte van de afvalrand in de Y richting aan de linkerzijde*)
	g_HMI_RCP_Parameters_Visu.rSizeTrimFront:=60;		(*grootte van de afvalrand in de Y richting aan de rechterzijde*)
	g_HMI_RCP_Parameters_Visu.rDiameterRound:=24;
	g_HMI_RCP_Parameters_Visu.rMidPosOffsetRound1X:= 0;		(* For round products *)
	g_HMI_RCP_Parameters_Visu.rMidPosOffsetRound1Y:= 0;		(* For round products *)
	g_HMI_RCP_Parameters_Visu.rMidPosOffsetRound2Y:= 0;		(* For round products *)
	g_HMI_RCP_Parameters_Visu.bTrianglesInTray:= FALSE;	(* For tray product *)
	g_HMI_RCP_Parameters_Visu.bUseRectanglesForTriangles:= FALSE;	(* For triangles only*)
	g_HMI_RCP_Parameters_Visu.bUseRectanglesInEight:= FALSE;	(* For triangles in tray only*)
	g_HMI_RCP_Parameters_Visu.bCutRoundInSequence	:=TRUE;
	g_HMI_RCP_Parameters_Visu.rPartSizeX	:= 50;	(* For triangles only *)
	g_HMI_RCP_Parameters_Visu.rPartSizeY := 50;	(* For triangles only *)
	g_HMI_RCP_Parameters_Visu.rShiftCompensation := 0;		(* For slab square only, compensation due to product shoved away during cutting (e.g. when product is slippery or frozen) *)
	g_HMI_RCP_Parameters_Visu.rSpeedTableXY := 100;	(* in % *)
	g_HMI_RCP_Parameters_Visu.rCleaningTimeUltrasonic	:= 5;		(* in sec *)
	g_HMI_RCP_Parameters_Visu.rCleaningTimeWater:= 5;		(* in sec *)
	g_HMI_RCP_Parameters_Visu.rCleaningTimeAir:= 5;		(* in sec *)
	g_HMI_RCP_Parameters_Visu.nCleanAfterNProd := 1;
	g_HMI_RCP_Parameters_Visu.nCleanProdOrCuts :=0;			(* Cleaning after number of products or after number of cuts. 0 = product, 1 = cuts *)
	g_HMI_RCP_Parameters_Visu.nCleanWithScraper:=1;			(* V10.01 Cleaning cycle with the use of *)
														(*        0 = Water and scraper *)
														(*        1 = Scraper only *)
														(*        2 = Water only *)

	g_HMI_RCP_Parameters_Visu.bMirrorDiagonals := FALSE;
END_IF');
%NETWORK
L_RecipeManager1(xEnable := TRUE, sDatabaseName := 'Recipes', sSelectedRecipeName := sSelectedRecipeName, xRecipe_Load := g_HMI_MachCommand.CMD.bLoadRecipe, xRecipe_New := g_HMI_MachCommand.CMD.bNewRecipe, xRecipe_Edit := g_HMI_MachCommand.CMD.bEditRecipe, xRecipe_Save := g_HMI_MachCommand.CMD.bSaveRecipe, xRecipe_Copy := g_HMI_MachCommand.CMD.bCopyRecipe, xRecipe_Delete := g_HMI_MachCommand.CMD.bDeleteRecipe, xRecipe_Update := g_HMI_MachCommand.CMD.bUpdateRecipe, scRecipeVisu := g_HMI_RCP_Parameters_Visu, scRecipePLC := g_HMI_RCP_Parameters, sRecipeNames => sRecipeNames, dwReturnValue => dwReturnValue);
%NETWORK
// Generate machinepar name based on system time.
GetDateAndTime(xExecute := g_HMI_MachCommand.CMD.bSaveMachPar, dtDateAndTime => dtDateAndTIme);
%NETWORK
ASSIGN(TO_STRING(dtDateAndTIme), Q => sDateAndTIme);
%NETWORK
ASSIGN(DELETE(STR := sDateAndTIme, LEN := 4, POS := 0), Q => sDateAndTIme1);
%NETWORK
ASSIGN(REPLACE(STR1 := sDateAndTIme1, STR2 := 'h', L := 1, P := 14), Q => sDateAndTIme2);
%NETWORK
ASSIGN(REPLACE(STR1 := sDateAndTIme2, STR2 := 'm', L := 1, P := 17), Q => sRecipeNamePar);
%NETWORK
EXECUTE(EN := TRUE, 'IF g_HMI_MachCommand.CMD.bSaveMachPar AND GetDateAndTime.xDone THEN
	sMachParName := sRecipeNamePar;
	bSavePars := TRUE;
	g_HMI_MachCommand.CMD.bSaveMachPar := FALSE;
END_IF');
%NETWORK
%NETWORK
L_MachParManager1(xEnable := TRUE, sDatabaseName := 'MachPar', sRecipeName := sMachParName, xRecipe_Delete := g_HMI_MachCommand.CMD.bDeleteMachPar, xRecipe_Load := g_HMI_MachCommand.CMD.bLoadMachPar, xRecipe_Save := bSaveParAs, xRecipe_SaveAs := bSavePars, sActiveRecipe := sActiveMachPar, sRecipeNames => sMachParNames, dwReturnValue => dwMachParReturnValue);

END_PROGRAM
